FUNCTION alg_g_algeb1: LREAL
VAR_INPUT
    state: STATE;
END_VAR

alg_g_algeb1 := (state.curTime) + (1.0);

END_FUNCTION

(* stored: ProductVersion 3.1.0.18, Version 1.1.0.1 *)
